TYPE StepStatus :
STRUCT
	status		: E_Result;
	elapsedTime : TIME;
END_STRUCT
END_TYPE

(* stored: Version 1.1.0.1, ProductVersion 3.1.4024.11
   DUT StepStatus: Id {99fb0db3-9288-4a62-a866-8e925fb082bf} *)
